// TIA Portal project "Bai 7" (V16)

(* hardware
DEVICE "S7-1200 station_1"  S7-1200 Station
   slot 0: "Rack_0"  S7-1200 Rack  Rack  V1.0
   slot 1: "PLC_1"  CPU 1214C DC/DC/DC  6ES7 214-1AG40-0XB0  V4.2
   slot 2: "DQ 16xRelay_1"  SM 1222 DQ16 x relay  6ES7 222-1HH32-0XB0  V2.0
*)

// ===== PLC "PLC_1"  CPU 1214C DC/DC/DC =====

VAR_GLOBAL   // PLC tag table "Default tag table"
   "Start" AT %I0.0 : Bool;
   "Quay_DC" AT %Q9.0 : Bool;
   "Khoan" AT %Q9.1 : Bool;
   "Tag_4" AT %Q9.5 : Bool;
   "Tag_5" AT %Q9.6 : Bool;
   "Tag_6" AT %M0.0 : Bool;
   "SQ1" AT %I0.3 : Bool;
   "Tag_8" AT %M1.1 : Bool;
   "Tag_9" AT %M1.2 : Bool;
   "Stop" AT %I0.1 : Bool;
   "Tag_11" AT %M1.3 : Bool;
   "Tag_12" AT %M0.1 : Bool;
   "Tag_13" AT %M0.2 : Bool;
   "Tag_1" AT %M1.4 : Bool;
   "Tag_2" AT %M1.7 : Bool;
   "Tag_10" AT %M1.0 : Bool;
   "Tag_14" AT %M0.7 : Bool;
   "SQ2" AT %I0.4 : Bool;
   "SQ3" AT %I0.5 : Bool;
   "Tag_16" AT %M0.3 : Bool;
   "Tag_17" AT %M0.4 : Bool;
   "KepPhoi" AT %Q9.2 : Bool;
   "Tag_3" AT %M0.5 : Bool;
   "Tag_7" AT %M0.6 : Bool;
END_VAR

// folder: System blocks/Program resources

DATA_BLOCK "T1"   // DB1
{ S7_Optimized_Access := 'TRUE' }
AUTHOR : Simatic
FAMILY : IEC
NAME : IEC_TMR
VERSION : 1.0
// stored: InstanceOfName IEC_TIMER
"IEC_TIMER"
BEGIN
END_DATA_BLOCK

DATA_BLOCK "T2"   // DB2
{ S7_Optimized_Access := 'TRUE' }
AUTHOR : Simatic
FAMILY : IEC
NAME : IEC_TMR
VERSION : 1.0
// stored: InstanceOfName IEC_TIMER
"IEC_TIMER"
BEGIN
END_DATA_BLOCK

DATA_BLOCK "T3"   // DB3
{ S7_Optimized_Access := 'TRUE' }
AUTHOR : Simatic
FAMILY : IEC
NAME : IEC_TMR
VERSION : 1.0
// stored: InstanceOfName IEC_TIMER
"IEC_TIMER"
BEGIN
END_DATA_BLOCK

DATA_BLOCK "T4"   // DB4
{ S7_Optimized_Access := 'TRUE' }
AUTHOR : Simatic
FAMILY : IEC
NAME : IEC_TMR
VERSION : 1.0
// stored: InstanceOfName IEC_TIMER
"IEC_TIMER"
BEGIN
END_DATA_BLOCK

DATA_BLOCK "T5"   // DB5
{ S7_Optimized_Access := 'TRUE' }
AUTHOR : Simatic
FAMILY : IEC
NAME : IEC_TMR
VERSION : 1.0
// stored: InstanceOfName IEC_TIMER
"IEC_TIMER"
BEGIN
END_DATA_BLOCK

DATA_BLOCK "T6"   // DB6
{ S7_Optimized_Access := 'TRUE' }
AUTHOR : Simatic
FAMILY : IEC
NAME : IEC_TMR
VERSION : 1.0
// stored: InstanceOfName IEC_TIMER
"IEC_TIMER"
BEGIN
END_DATA_BLOCK

// folder: (top level)

ORGANIZATION_BLOCK "Main"   // OB1, LAD, ProgramCycle
TITLE = "Main Program Sweep (Cycle)"
{ S7_Optimized_Access := 'TRUE' }
VERSION : 0.1
   VAR_INPUT
      Initial_Call : Bool;   // Initial call of this OB
      Remanence : Bool;   // =True, if remanent data are available
   END_VAR
   VAR_TEMP   // added for the SCL form of the ladder/FBD networks
      _w1 : Bool;
   END_VAR
BEGIN

REGION Network 1
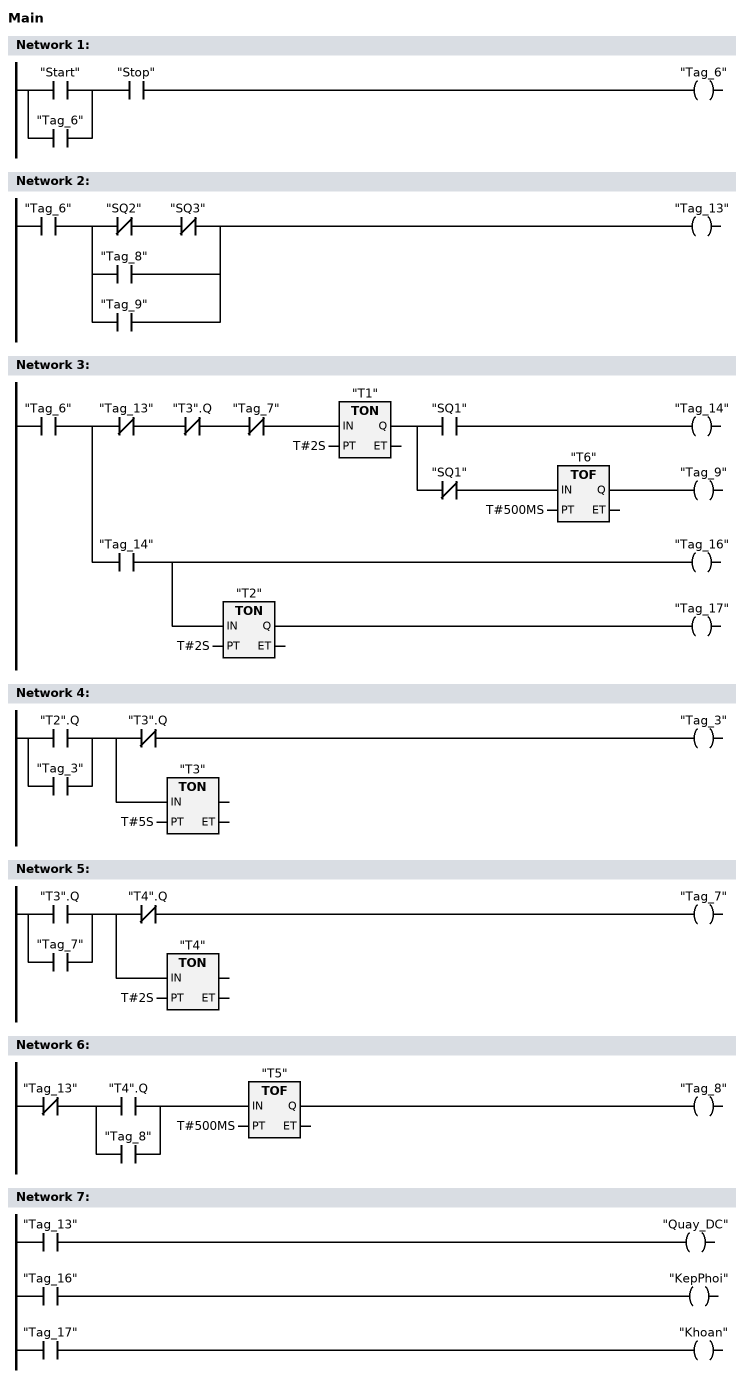
   RUNG wire#powerrail
      Contact( "Start" )
      wire#w1
      Contact( "Stop" )
      Coil( "Tag_6" )
   END_RUNG
   RUNG wire#powerrail
      Contact( "Tag_6" )
   END_RUNG wire#w1
   // the same network as SCL:
   "Tag_6" := ("Start" OR "Tag_6") AND "Stop";
END_REGION

REGION Network 2
   RUNG wire#powerrail
      Contact( "Tag_6" )
      wire#w1
      I_Contact( "SQ2" )
      I_Contact( "SQ3" )
      wire#w2
      Coil( "Tag_13" )
   END_RUNG
   RUNG wire#w1
      Contact( "Tag_8" )
   END_RUNG wire#w2
   RUNG wire#w1
      Contact( "Tag_9" )
   END_RUNG wire#w2
   // the same network as SCL:
   "Tag_13" := "Tag_6" AND ((NOT "SQ2" AND NOT "SQ3") OR "Tag_8" OR "Tag_9");
END_REGION

REGION Network 3
   "T1".TON(IN := "Tag_6" AND NOT "Tag_13" AND NOT "T3".Q AND NOT "Tag_7", PT := T#2S);
   "Tag_14" := "T1".Q AND "SQ1";
   "T6".TOF(IN := "T1".Q AND NOT "SQ1", PT := T#500MS);
   "Tag_9" := "T6".Q;
   "Tag_16" := "Tag_6" AND "Tag_14";
   "T2".TON(IN := "Tag_16", PT := T#2S);
   "Tag_17" := "T2".Q;
END_REGION

REGION Network 4
   #_w1 := "T2".Q OR "Tag_3";
   "Tag_3" := #_w1 AND NOT "T3".Q;
   "T3".TON(IN := #_w1, PT := T#5S);
END_REGION

REGION Network 5
   #_w1 := "T3".Q OR "Tag_7";
   "Tag_7" := #_w1 AND NOT "T4".Q;
   "T4".TON(IN := #_w1, PT := T#2S);
END_REGION

REGION Network 6
   "T5".TOF(IN := NOT "Tag_13" AND ("T4".Q OR "Tag_8"), PT := T#500MS);
   "Tag_8" := "T5".Q;
END_REGION

REGION Network 7
   RUNG wire#powerrail
      Contact( "Tag_13" )
      Coil( "Quay_DC" )
   END_RUNG
   RUNG wire#powerrail
      Contact( "Tag_16" )
      Coil( "KepPhoi" )
   END_RUNG
   RUNG wire#powerrail
      Contact( "Tag_17" )
      Coil( "Khoan" )
   END_RUNG
   // the same network as SCL:
   "Quay_DC" := "Tag_13";
   "KepPhoi" := "Tag_16";
   "Khoan" := "Tag_17";
END_REGION
END_ORGANIZATION_BLOCK